// TIA Portal V20 export
DATA_BLOCK "OPCUA"   // DB900
TITLE = INTERFACE
{ S7_Optimized_Access := 'FALSE' }
AUTHOR : HYUNDAI-MOVEX
FAMILY : LGR
VERSION : 0.1
// stored: AutoNumber false, DBAccessibleFromOPCUA true, DBAccessibleFromWebserver false, IsOnlyStoredInLoadMemory false, IsWriteProtectedInAS false
   VAR
      CMD : "LGR_Interface_GR_Command";
      STAT : "LGR_Interface_GR_Status";
   END_VAR
BEGIN
END_DATA_BLOCK
